INTERFACE ITrafficLight

PROPERTY CurrentState  : E_LightState
GET
END_GET
END_PROPERTY

METHOD Cycle
VAR
END_VAR
END_METHOD

END_INTERFACE

(* stored: Version 1.1.0.1, ProductVersion 3.1.4024.12
   Itf ITrafficLight: Id {b2039307-2a7b-4887-9fed-80e45ee06bce}
   Property CurrentState: Id {c01ada10-c8cc-48ae-9c46-da2e0692e2de}
   Get Get: Id {ad11bb5a-8608-41b6-baaa-619ecae7a69e}
   Method Cycle: Id {892fb504-fa89-4974-8c21-d7396bf0d00e} *)
